(* CODESYS project Control.gvl.xml

Project tree, tasks and I/O mapping:
  global variables Control
*)

// Control
{attribute 'qualified_only'}
VAR_GLOBAL
	FaultReset: FaultReset;
	Logger: Logger;
	ManualControl: ManualControl;
	LoadDefaults: BOOL;
END_VAR
